{attribute addProperty BoxType "EJ2522-0000-0022"}
{attribute addProperty Id "PTO_Status_ChannelAT %I*ARRAY[0..1] OF PTO_Status_Channel_B9BB57FE3240ENC_Status_ChannelAT %I*ARRAY[0..2] OF ENC_Status_Channel_D7F8917396120PTO_Control_Channel_1AT %Q*PTO_Control_Channel_0A6210C33240PTO_Target_Channel_1AT %Q*PTO_Target_Channel_3945899C3240PTO_Control_Channel_2AT %Q*PTO_Control_Channel_0A6210C33240PTO_Target_Channel_2AT %Q*PTO_Target_Channel_3945899C3240ENC_Control_ChannelAT %Q*ARRAY[0..2] OF ENC_Control_Channel_8309D56E96120WcStateAT %I*WcState_98A4DF7520.250InfoDataAT %I*InfoData_BC63D37F80100"}
{attribute addProperty CRC "1184876195"}
{attribute addProperty SizeInBites "434"}
{attribute addProperty SizeInBytes "54.25"}
TYPE EJ2522_58A1BC1F :
STRUCT
	{attribute addProperty Name "PTO_Status_Channel"}
	PTO_Status_Channel : ARRAY[0..1] OF PTO_Status_Channel_B9BB57FE;
	{attribute addProperty Name "ENC_Status_Channel"}
	ENC_Status_Channel : ARRAY[0..2] OF ENC_Status_Channel_D7F89173;
	{attribute addProperty Name "PTO_Control_Channel_1"}
	PTO_Control_Channel_1 : PTO_Control_Channel_0A6210C3;
	{attribute addProperty Name "PTO_Target_Channel_1"}
	PTO_Target_Channel_1 : PTO_Target_Channel_3945899C;
	{attribute addProperty Name "PTO_Control_Channel_2"}
	PTO_Control_Channel_2 : PTO_Control_Channel_0A6210C3;
	{attribute addProperty Name "PTO_Target_Channel_2"}
	PTO_Target_Channel_2 : PTO_Target_Channel_3945899C;
	{attribute addProperty Name "ENC_Control_Channel"}
	ENC_Control_Channel : ARRAY[0..2] OF ENC_Control_Channel_8309D56E;
	{attribute addProperty Name "WcState"}
	WcState : WcState_98A4DF75;
	{attribute addProperty Name "InfoData"}
	InfoData : InfoData_BC63D37F;
END_STRUCT
END_TYPE

(* stored: Version 1.2.0.0, ProductVersion 3.1.4024.9
   DUT EJ2522_58A1BC1F: Id {c0c448c3-3942-44ba-abd6-fa64071c4e08} *)
